# EPICS autosave request: ipApp/Db/PHD2000_settings.req
# CPSyringe_settings.req
#
# Autosave file for Harvard Apparatus syringe pump
#
# Mark Rivers
# November 23, 2013

$(P)$(R)ReadSettings.SCAN
$(P)$(R)Mode
$(P)$(R)Direction
$(P)$(R)Diameter
$(P)$(R)InfusionRate
$(P)$(R)WithdrawalRate
$(P)$(R)InfusionVolume
